(* PLC project v0.6.04_CycleSemiAuto.project, CODESYS CODESYS V3.5 SP19 Patch 1 *)
(* stored: creationDateTime 2026-08-11T14:02:33.683303, modificationDateTime 2026-08-11T14:02:33.683303 *)

(* ═══════════════════════════════════════════════════════════════ 🎮 ST_TranslationCmd — Commandes IHM pour la Translation M3 ─────────────────────────────────────────────────────────────── 🎨 Destiné au pilotage de la translation M3 depuis l'IHM. 📄 2026-07-24 : Initialized protège SetFreq_Hz (seul réglage à survivre au reboot), sans pont générique pour ne jamais persister BtnFwd/BtnRev. ═══════════════════════════════════════════════════════════════ *)
TYPE ST_TranslationCmd : STRUCT
  SelPositioning : BOOL;  (* 🎯 TRUE = positionneur sur SelTarget ; FALSE = jog libre *)
  SelTarget : INT;  (* 🔢 Numéro de la cible de position sélectionnée *)
  BtnFwd : BOOL;  (* ↔️ Requête marche avant (→ Trémie), pilotage IHM exclusif *)
  BtnRev : BOOL;  (* ↔️ Requête marche arrière (→ Maintenance), pilotage IHM exclusif *)
  SetFreq_Hz : REAL;  (* 🎯 Consigne fréquence manuelle [Hz], limitée par PRG_10_Outputs_LD *)
  InvertDirection : BOOL;  (* 🔀 2026-08-06 : TglJoystickMaster PAR AXE supprimé (doublon) — un seul switch machine : GVL_IHM.Modes.Cmd.TglJoystickMaster (ST_ModesCmd), applicable à M1/M2 ET M3. 🔄 TRUE = inverse Fwd→Maintenance / Rev→Trémie (mise en service) *)
  TglMaintenanceZoneAccess : BOOL;  (* 🆕 2026-08-06 : autorisation CONSCIENTE zone Maintenance, EN PLUS de MAINT_N2 (Auth.MaintenanceM3TargetEnable) *)
  Initialized : BOOL := FALSE;  (* 🚦 TRUE = SetFreq_Hz restauré depuis GVL_PERSISTENT ce boot *)
END_STRUCT;
END_TYPE
